{attribute addProperty BoxType "EM7004-0000-9995"}
{attribute addProperty Id "InputAT %I*ARRAY[0 ..15] OF BOOL128160"}
{attribute addProperty CRC "1547216551"}
{attribute addProperty SizeInBites "128"}
{attribute addProperty SizeInBytes "16"}
TYPE Digital_42B6F5B2 :
STRUCT
	{attribute addProperty Name "Input"}
	Input AT %I* : ARRAY[0 ..15] OF BOOL;
END_STRUCT
END_TYPE

(* stored: Version 1.2.0.0, ProductVersion 3.1.4024.9
   DUT Digital_42B6F5B2: Id {e4e4ffae-fe7d-466e-a8c4-dfe91e2057aa} *)
